TYPE st_ListRunCore :
STRUCT
	ListRunCore : ARRAY[0..12] OF st_FlowBaseCore;
END_STRUCT
END_TYPE

(* stored: Version 1.1.0.1, ProductVersion 3.1.4024.13
   DUT st_ListRunCore: Id {affdd455-49bb-4846-bb84-e4ed20855371} *)
